FUNCTION Update_Command_State : BOOL
VAR_INPUT
	Camera : REFERENCE TO Cognex_Camera;
END_VAR
VAR
END_VAR

IF Camera.CommandState = Command_State.Wate THEN
	IF Camera.Inspection.COmmandCompleted THEN
		Camera.CommandState := Command_State.Complete;
		Camera.Inspection.ExecuteCommand := FALSE;
	ELSIF Camera.Inspection.CommandFailed THEN
		Camera.CommandState := Command_State.Error;
		Camera.CameraState := Camera_State.Error;
		Camera.Inspection.ExecuteCommand := FALSE;
		CASE Camera.Inspection.ErrorCode OF
			16#0100: // Trigger set while disabeld
				Camera.Error := Camera_Error.Trigger_Set_While_disabeld;
			16#0101: // trigger set while offline
				Camera.Error := Camera_Error.Trigger_Set_While_Offline;
			16#0400: // already executing error
				Camera.Error := Camera_Error.Already_Executing;
			16#0401: // job load requeted while online
				Camera.Error := Camera_Error.Job_Load_Requested_While_Online;
			16#0402: // job load requested does not exist on the camera
				Camera.Error := Camera_Error.Job_Does_Not_Exist;
		END_CASE
		RETURN;
	END_IF
ELSIF Camera.CommandState = Command_State.Error THEN
	Camera.CommandState := Command_State.Error;
	Camera.CameraState := Camera_State.Error;
	CASE Camera.Inspection.ErrorCode OF
		16#0100: // Trigger set while disabeld
			Camera.Error := Camera_Error.Trigger_Set_While_disabeld;
		16#0101: // trigger set while offline
			Camera.Error := Camera_Error.Trigger_Set_While_Offline;
		16#0400: // already executing error
			Camera.Error := Camera_Error.Already_Executing;
		16#0401: // job load requeted while online
			Camera.Error := Camera_Error.Job_Load_Requested_While_Online;
		16#0402: // job load requested does not exist on the camera
			Camera.Error := Camera_Error.Job_Does_Not_Exist;
	END_CASE
	RETURN;
ELSE
	Camera.CommandState := Command_State.Error;
	Camera.Error := Camera_Error.StateError;
	RETURN;
END_IF

END_FUNCTION

(* stored: Version 1.1.0.1, ProductVersion 3.1.4024.10
   POU Update_Command_State: Id {37a8c9d7-ccce-4f74-b94a-86dc9c36ae06}, SpecialFunc None *)
